(* Logix 5000 project; controller GEA_Test_Chamber vendor 1 type 14 code 196 rev 32.14; software revision 32.04; part 9 of 11 *)
(* tags used below, declared in another part *)
   Act_Time : DINT[7];
   bPulse05Hz : BOOL;
   bPulse0_1Hz : BOOL;
   bPulse10Hz : BOOL;
   bPulse1Hz : BOOL;
   bPulse1min : BOOL;
   Counter : COUNTER[20];
   LDO_LabView_Comm_OK : BOOL;
   LDO_Oil_Step : INT;
   LDO_Step : INT;
   New_Time : BOOL;
   Oil_spray_08_ccmin : BOOL;
   Oil_spray_11_ccmin : BOOL;
   Oil_spray_133_ccmin : BOOL;
   Pulse : BOOL[32];
   Step_10_Done : BOOL;
   Step_20_Done : BOOL;
   Step_25_Done : BOOL;
   Step_30_Done : BOOL;
   Step_40_Done : BOOL;
   Step_5_Done : BOOL;
   T_Diff_10 : DINT;
   T_Diff_20 : DINT;
   T_Diff_25 : DINT;
   T_Diff_30 : DINT;
   T_Diff_40 : DINT;
   T_Diff_5 : DINT;
   T_Diff_Step10 : T_DIFF;
   T_Diff_Step20 : T_DIFF;
   T_Diff_Step25 : T_DIFF;
   T_Diff_Step30 : T_DIFF;
   T_Diff_Step40 : T_DIFF;
   T_Diff_Step5 : T_DIFF;
   Time_Step_10 : DINT[7];
   Time_Step_20 : DINT[7];
   Time_Step_25 : DINT[7];
   Time_Step_30 : DINT[7];
   Time_Step_40 : DINT[7];
   Time_Step_5 : DINT[7];
   tof0_1sPulse : TIMER;
   tof10sPulse : TIMER;
   tof1sPulse : TIMER;
   tof2sPulse : TIMER;
   tof30sPulse : TIMER;
   ton0_1sPulse : TIMER;
   ton10sPulse : TIMER;
   ton1sPulse : TIMER;
   ton2sPulse : TIMER;
   ton30sPulse : TIMER;
   TON_LifeBit_OFF : TIMER;
   TON_LifeBit_ON : TIMER;
   Control_Off : BOOL;
   FVIR_LabView_Control : INT;
   LDO_Error_MSG : INT;
   LDO_LabView_Control : INT;
   LDO_LabView_Control2 : INT;
   LDO_LabView_Status : INT;
   LDO_Reset_CNT_inprogress : BOOL;
   Modbus_LabView_Data : raC_UDT_ModbusServerData;
   Oil_inj_08_Cnt : COUNTER;
   Oil_inj_11_Cnt : COUNTER;
   Oil_inj_133_Cnt : COUNTER;
   Output_LDO : Output_LDO;
(* LDO_Chamber, continued *)

ROUTINE LDO_Main   (* ladder *)
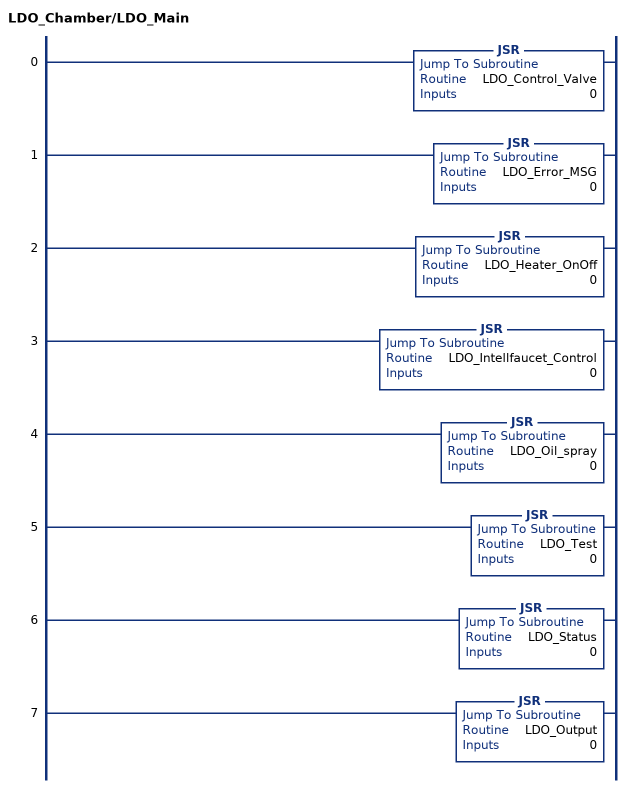
   0: JSR(LDO_Control_Valve,0);
   1: JSR(LDO_Error_MSG,0);
   2: JSR(LDO_Heater_OnOff,0);
   3: JSR(LDO_Intellfaucet_Control,0);
   4: JSR(LDO_Oil_spray,0);
   5: JSR(LDO_Test,0);
   6: JSR(LDO_Status,0);
   7: JSR(LDO_Output,0);
END_ROUTINE

ROUTINE LDO_Oil_spray   (* ladder *)
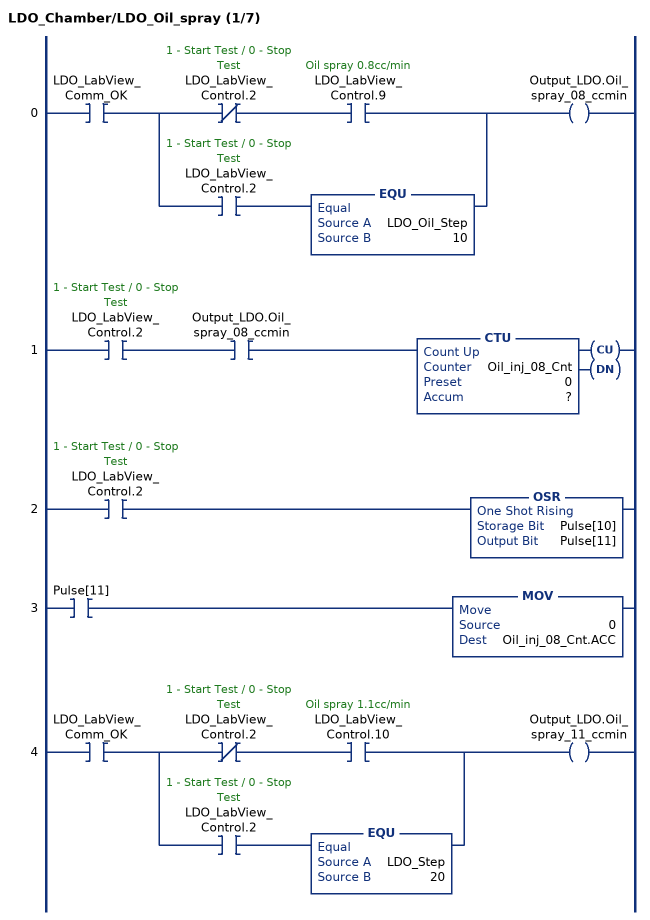
   0: XIC(LDO_LabView_Comm_OK)[XIO(LDO_LabView_Control.2) XIC(LDO_LabView_Control.9) ,XIC(LDO_LabView_Control.2) EQU(LDO_Oil_Step,10) ]OTE(Output_LDO.Oil_spray_08_ccmin);
   1: XIC(LDO_LabView_Control.2)XIC(Output_LDO.Oil_spray_08_ccmin)CTU(Oil_inj_08_Cnt,?,?);
   2: XIC(LDO_LabView_Control.2)OSR(Pulse[10],Pulse[11]);
   3: XIC(Pulse[11])MOV(0,Oil_inj_08_Cnt.ACC);
   4: XIC(LDO_LabView_Comm_OK)[XIO(LDO_LabView_Control.2) XIC(LDO_LabView_Control.10) ,XIC(LDO_LabView_Control.2) EQU(LDO_Step,20) ]OTE(Output_LDO.Oil_spray_11_ccmin);
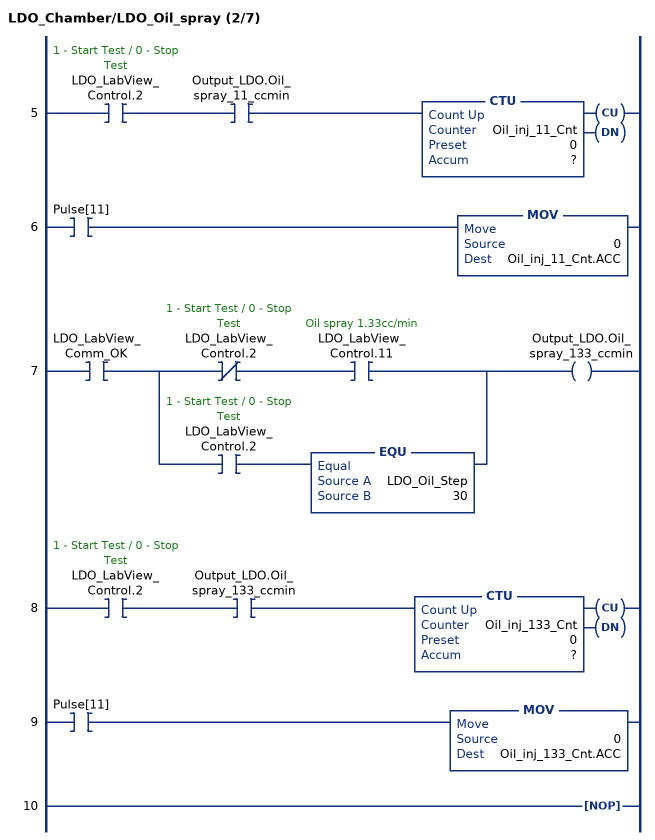
   5: XIC(LDO_LabView_Control.2)XIC(Output_LDO.Oil_spray_11_ccmin)CTU(Oil_inj_11_Cnt,?,?);
   6: XIC(Pulse[11])MOV(0,Oil_inj_11_Cnt.ACC);
   7: XIC(LDO_LabView_Comm_OK)[XIO(LDO_LabView_Control.2) XIC(LDO_LabView_Control.11) ,XIC(LDO_LabView_Control.2) EQU(LDO_Oil_Step,30) ]OTE(Output_LDO.Oil_spray_133_ccmin);
   8: XIC(LDO_LabView_Control.2)XIC(Output_LDO.Oil_spray_133_ccmin)CTU(Oil_inj_133_Cnt,?,?);
   9: XIC(Pulse[11])MOV(0,Oil_inj_133_Cnt.ACC);
   10: NOP();
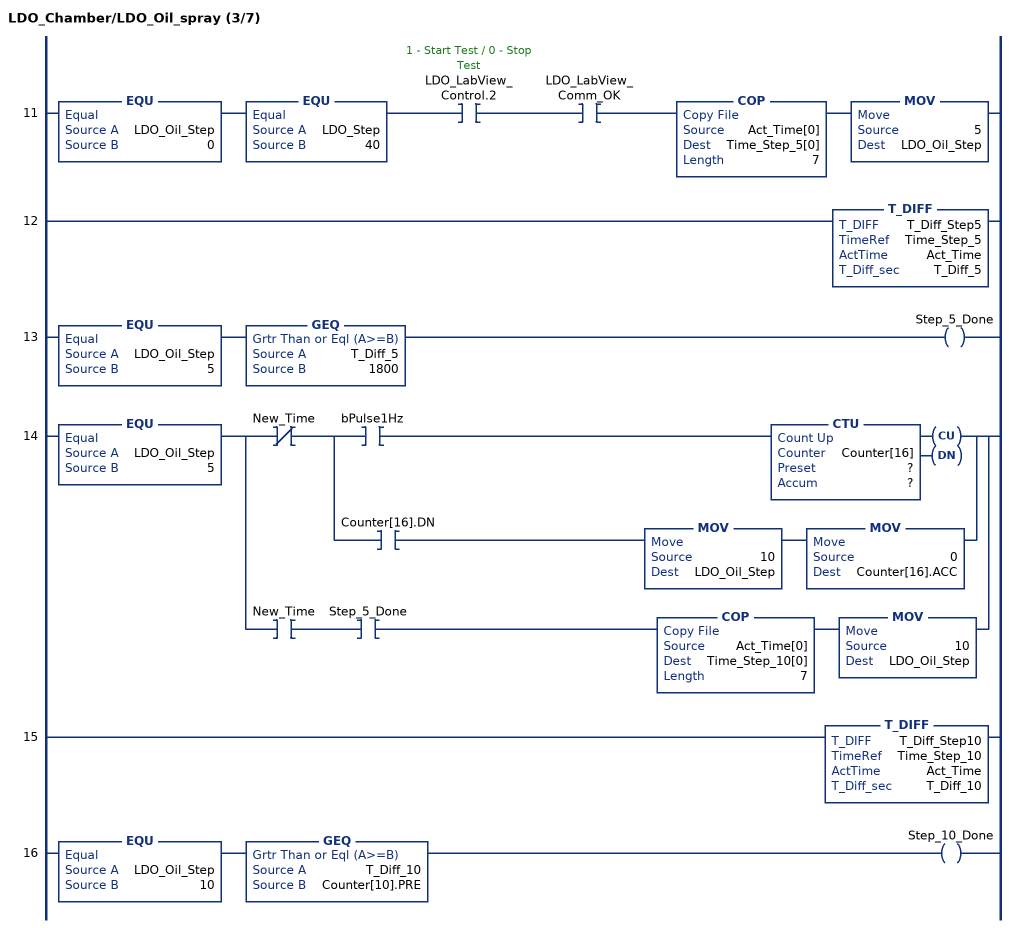
   11: EQU(LDO_Oil_Step,0)EQU(LDO_Step,40)XIC(LDO_LabView_Control.2)XIC(LDO_LabView_Comm_OK)COP(Act_Time[0],Time_Step_5[0],7)MOV(5,LDO_Oil_Step);
   12: T_DIFF(T_Diff_Step5,Time_Step_5,Act_Time,T_Diff_5);
   13: EQU(LDO_Oil_Step,5)GEQ(T_Diff_5,1800)OTE(Step_5_Done);
   14: EQU(LDO_Oil_Step,5)[XIO(New_Time) [XIC(bPulse1Hz) CTU(Counter[16],?,?) ,XIC(Counter[16].DN) MOV(10,LDO_Oil_Step) MOV(0,Counter[16].ACC) ] ,XIC(New_Time) XIC(Step_5_Done) COP(Act_Time[0],Time_Step_10[0],7) MOV(10,LDO_Oil_Step) ];
   15: T_DIFF(T_Diff_Step10,Time_Step_10,Act_Time,T_Diff_10);
   16: EQU(LDO_Oil_Step,10)GEQ(T_Diff_10,Counter[10].PRE)OTE(Step_10_Done);
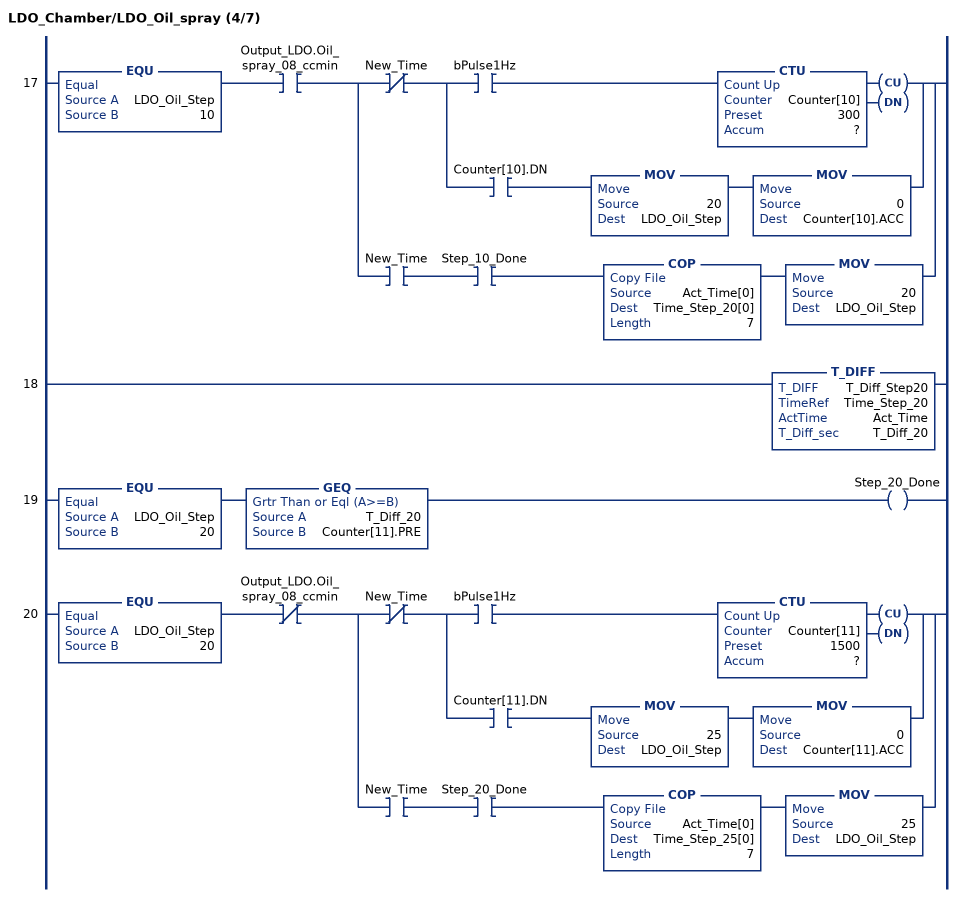
   17: EQU(LDO_Oil_Step,10)XIC(Output_LDO.Oil_spray_08_ccmin)[XIO(New_Time) [XIC(bPulse1Hz) CTU(Counter[10],?,?) ,XIC(Counter[10].DN) MOV(20,LDO_Oil_Step) MOV(0,Counter[10].ACC) ] ,XIC(New_Time) XIC(Step_10_Done) COP(Act_Time[0],Time_Step_20[0],7) MOV(20,LDO_Oil_Step) ];
   18: T_DIFF(T_Diff_Step20,Time_Step_20,Act_Time,T_Diff_20);
   19: EQU(LDO_Oil_Step,20)GEQ(T_Diff_20,Counter[11].PRE)OTE(Step_20_Done);
   20: EQU(LDO_Oil_Step,20)XIO(Output_LDO.Oil_spray_08_ccmin)[XIO(New_Time) [XIC(bPulse1Hz) CTU(Counter[11],?,?) ,XIC(Counter[11].DN) MOV(25,LDO_Oil_Step) MOV(0,Counter[11].ACC) ] ,XIC(New_Time) XIC(Step_20_Done) COP(Act_Time[0],Time_Step_25[0],7) MOV(25,LDO_Oil_Step) ];
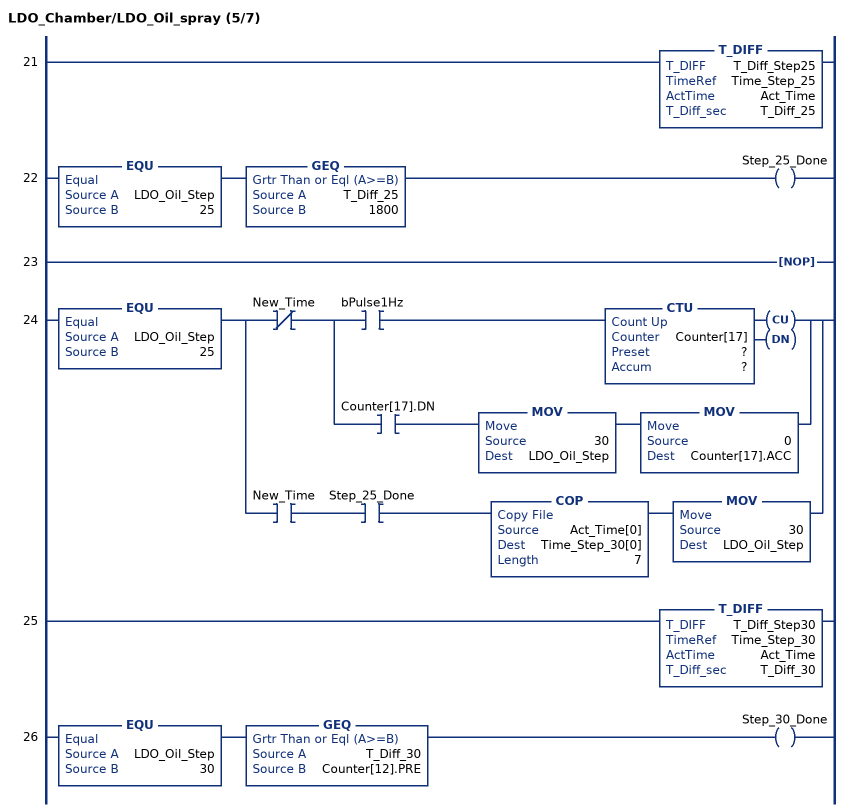
   21: T_DIFF(T_Diff_Step25,Time_Step_25,Act_Time,T_Diff_25);
   22: EQU(LDO_Oil_Step,25)GEQ(T_Diff_25,1800)OTE(Step_25_Done);
   23: NOP();
   24: EQU(LDO_Oil_Step,25)[XIO(New_Time) [XIC(bPulse1Hz) CTU(Counter[17],?,?) ,XIC(Counter[17].DN) MOV(30,LDO_Oil_Step) MOV(0,Counter[17].ACC) ] ,XIC(New_Time) XIC(Step_25_Done) COP(Act_Time[0],Time_Step_30[0],7) MOV(30,LDO_Oil_Step) ];
   25: T_DIFF(T_Diff_Step30,Time_Step_30,Act_Time,T_Diff_30);
   26: EQU(LDO_Oil_Step,30)GEQ(T_Diff_30,Counter[12].PRE)OTE(Step_30_Done);
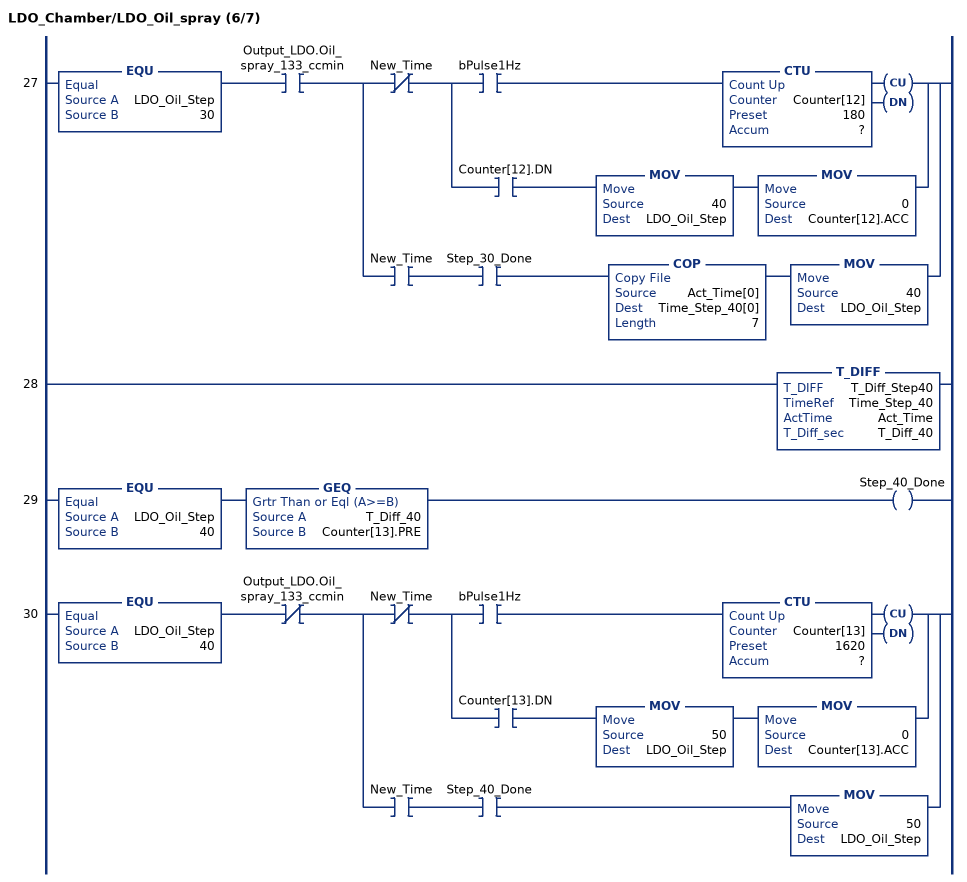
   27: EQU(LDO_Oil_Step,30)XIC(Output_LDO.Oil_spray_133_ccmin)[XIO(New_Time) [XIC(bPulse1Hz) CTU(Counter[12],?,?) ,XIC(Counter[12].DN) MOV(40,LDO_Oil_Step) MOV(0,Counter[12].ACC) ] ,XIC(New_Time) XIC(Step_30_Done) COP(Act_Time[0],Time_Step_40[0],7) MOV(40,LDO_Oil_Step) ];
   28: T_DIFF(T_Diff_Step40,Time_Step_40,Act_Time,T_Diff_40);
   29: EQU(LDO_Oil_Step,40)GEQ(T_Diff_40,Counter[13].PRE)OTE(Step_40_Done);
   30: EQU(LDO_Oil_Step,40)XIO(Output_LDO.Oil_spray_133_ccmin)[XIO(New_Time) [XIC(bPulse1Hz) CTU(Counter[13],?,?) ,XIC(Counter[13].DN) MOV(50,LDO_Oil_Step) MOV(0,Counter[13].ACC) ] ,XIC(New_Time) XIC(Step_40_Done) MOV(50,LDO_Oil_Step) ];
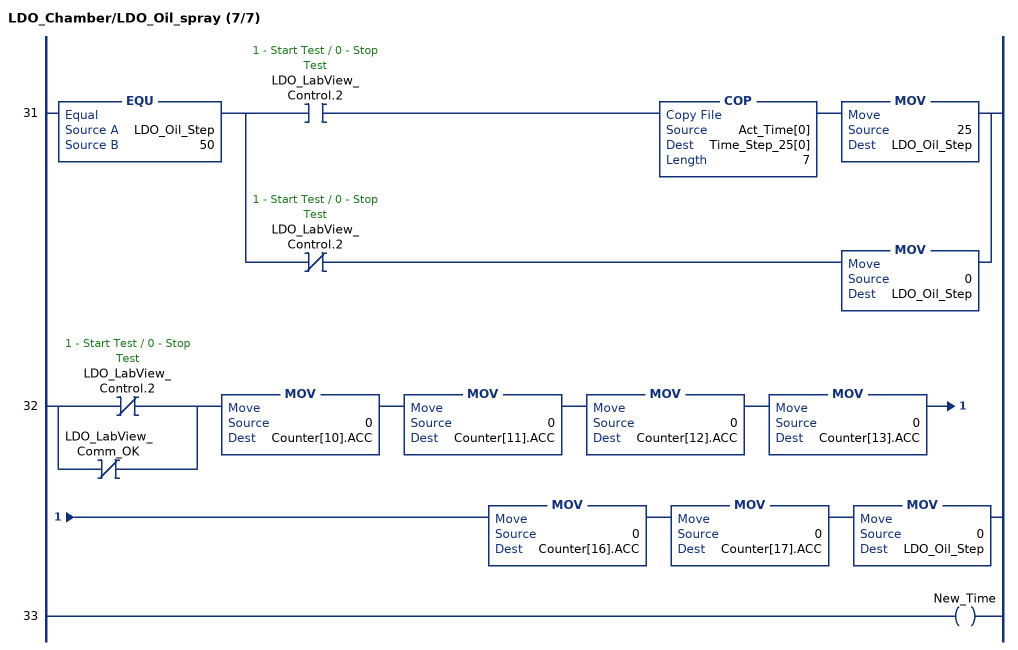
   31: EQU(LDO_Oil_Step,50)[XIC(LDO_LabView_Control.2) COP(Act_Time[0],Time_Step_25[0],7) MOV(25,LDO_Oil_Step) ,XIO(LDO_LabView_Control.2) MOV(0,LDO_Oil_Step) ];
   32: [XIO(LDO_LabView_Control.2) ,XIO(LDO_LabView_Comm_OK) ]MOV(0,Counter[10].ACC)MOV(0,Counter[11].ACC)MOV(0,Counter[12].ACC)MOV(0,Counter[13].ACC)MOV(0,Counter[16].ACC)MOV(0,Counter[17].ACC)MOV(0,LDO_Oil_Step);
   33: OTE(New_Time);
END_ROUTINE

ROUTINE LDO_Output   (* ladder *)
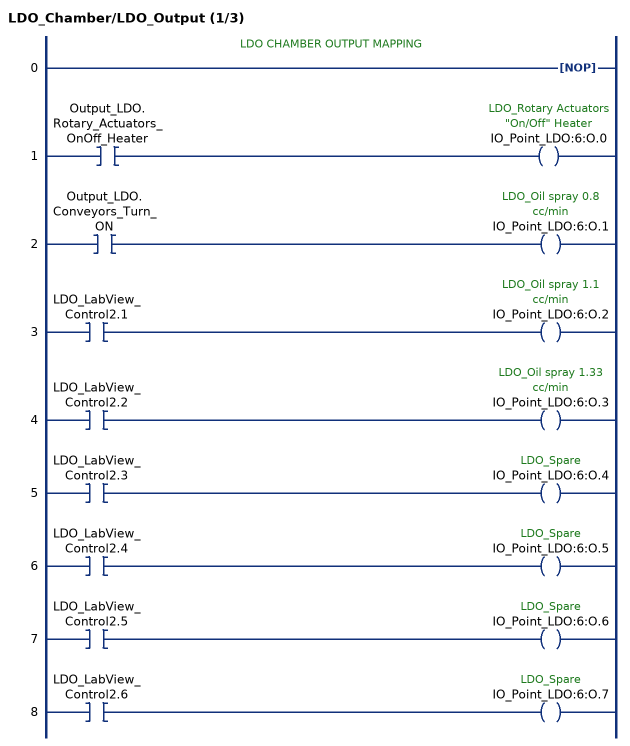
   // LDO CHAMBER OUTPUT MAPPING
   0: NOP();
   1: XIC(Output_LDO.Rotary_Actuators_OnOff_Heater)OTE(IO_Point_LDO:6:O.0);
   2: XIC(Output_LDO.Conveyors_Turn_ON)OTE(IO_Point_LDO:6:O.1);
   3: XIC(LDO_LabView_Control2.1)OTE(IO_Point_LDO:6:O.2);
   4: XIC(LDO_LabView_Control2.2)OTE(IO_Point_LDO:6:O.3);
   5: XIC(LDO_LabView_Control2.3)OTE(IO_Point_LDO:6:O.4);
   6: XIC(LDO_LabView_Control2.4)OTE(IO_Point_LDO:6:O.5);
   7: XIC(LDO_LabView_Control2.5)OTE(IO_Point_LDO:6:O.6);
   8: XIC(LDO_LabView_Control2.6)OTE(IO_Point_LDO:6:O.7);
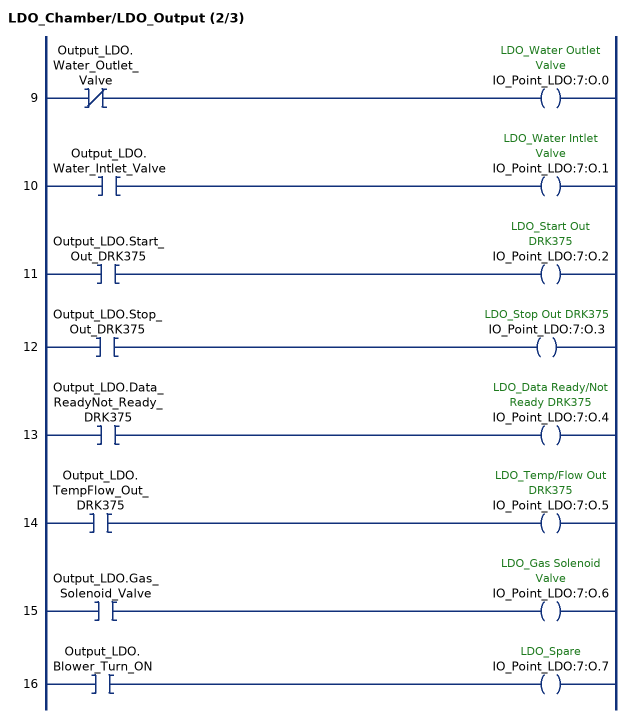
   9: XIO(Output_LDO.Water_Outlet_Valve)OTE(IO_Point_LDO:7:O.0);
   10: XIC(Output_LDO.Water_Intlet_Valve)OTE(IO_Point_LDO:7:O.1);
   11: XIC(Output_LDO.Start_Out_DRK375)OTE(IO_Point_LDO:7:O.2);
   12: XIC(Output_LDO.Stop_Out_DRK375)OTE(IO_Point_LDO:7:O.3);
   13: XIC(Output_LDO.Data_ReadyNot_Ready_DRK375)OTE(IO_Point_LDO:7:O.4);
   14: XIC(Output_LDO.TempFlow_Out_DRK375)OTE(IO_Point_LDO:7:O.5);
   15: XIC(Output_LDO.Gas_Solenoid_Valve)OTE(IO_Point_LDO:7:O.6);
   16: XIC(Output_LDO.Blower_Turn_ON)OTE(IO_Point_LDO:7:O.7);
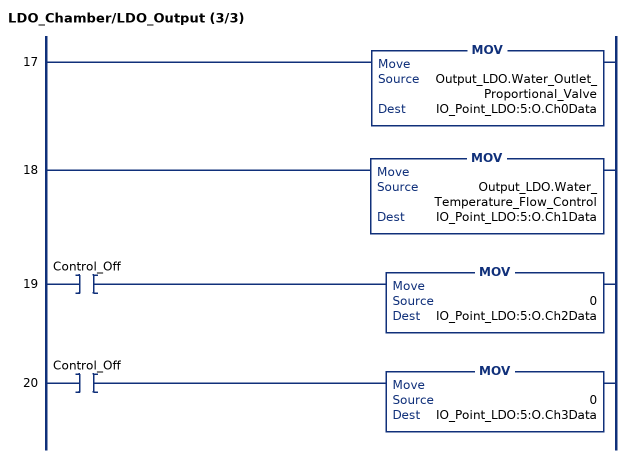
   17: MOV(Output_LDO.Water_Outlet_Proportional_Valve,IO_Point_LDO:5:O.Ch0Data);
   18: MOV(Output_LDO.Water_Temperature_Flow_Control,IO_Point_LDO:5:O.Ch1Data);
   19: XIC(Control_Off)MOV(0,IO_Point_LDO:5:O.Ch2Data);
   20: XIC(Control_Off)MOV(0,IO_Point_LDO:5:O.Ch3Data);
END_ROUTINE

ROUTINE LDO_Status   (* ladder *)
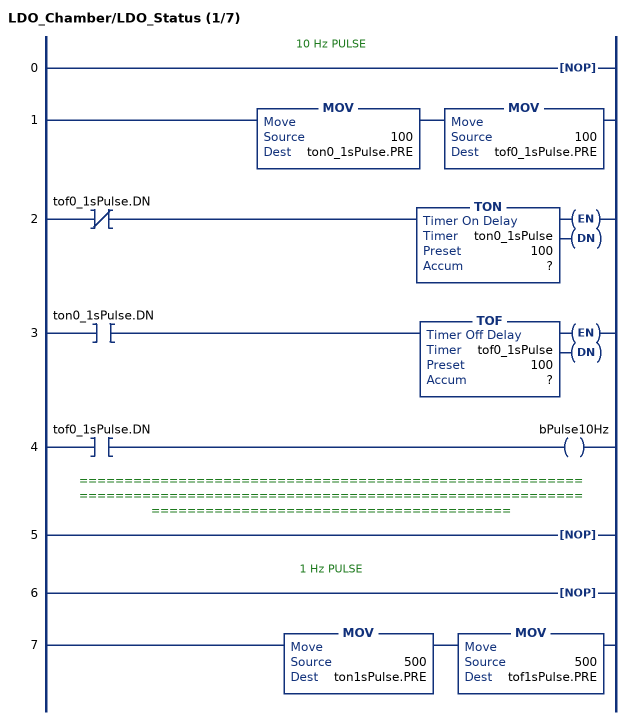
   // 10 Hz PULSE
   0: NOP();
   1: MOV(100,ton0_1sPulse.PRE)MOV(100,tof0_1sPulse.PRE);
   2: XIO(tof0_1sPulse.DN)TON(ton0_1sPulse,?,?);
   3: XIC(ton0_1sPulse.DN)TOF(tof0_1sPulse,?,?);
   4: XIC(tof0_1sPulse.DN)OTE(bPulse10Hz);
   // ========================================================================================================================================================
   5: NOP();
   // 1 Hz PULSE
   6: NOP();
   7: MOV(500,ton1sPulse.PRE)MOV(500,tof1sPulse.PRE);
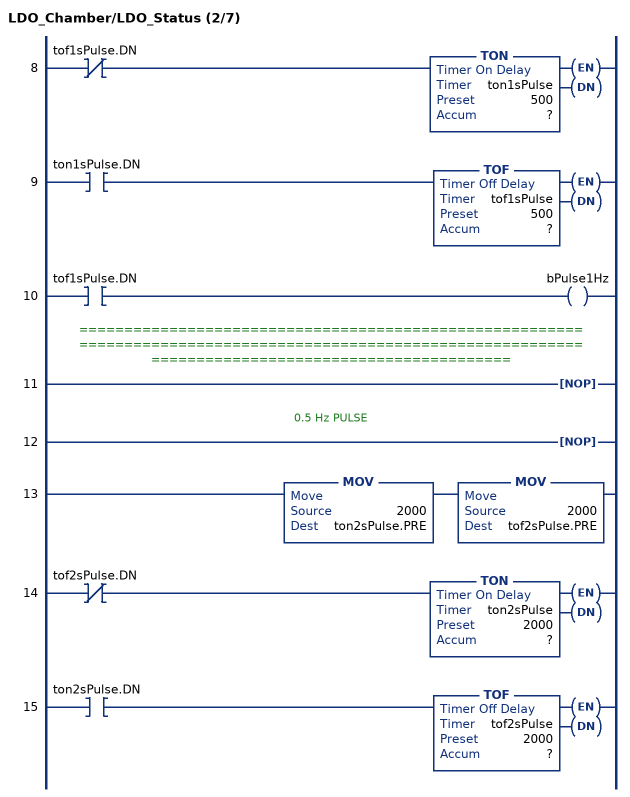
   8: XIO(tof1sPulse.DN)TON(ton1sPulse,?,?);
   9: XIC(ton1sPulse.DN)TOF(tof1sPulse,?,?);
   10: XIC(tof1sPulse.DN)OTE(bPulse1Hz);
   // ========================================================================================================================================================
   11: NOP();
   // 0.5 Hz PULSE
   12: NOP();
   13: MOV(2000,ton2sPulse.PRE)MOV(2000,tof2sPulse.PRE);
   14: XIO(tof2sPulse.DN)TON(ton2sPulse,?,?);
   15: XIC(ton2sPulse.DN)TOF(tof2sPulse,?,?);
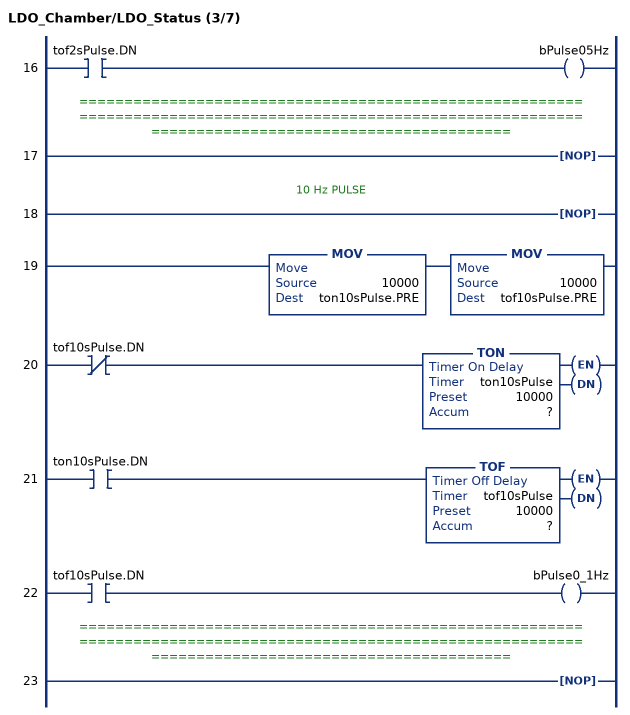
   16: XIC(tof2sPulse.DN)OTE(bPulse05Hz);
   // ========================================================================================================================================================
   17: NOP();
   // 10 Hz PULSE
   18: NOP();
   19: MOV(10000,ton10sPulse.PRE)MOV(10000,tof10sPulse.PRE);
   20: XIO(tof10sPulse.DN)TON(ton10sPulse,?,?);
   21: XIC(ton10sPulse.DN)TOF(tof10sPulse,?,?);
   22: XIC(tof10sPulse.DN)OTE(bPulse0_1Hz);
   // ========================================================================================================================================================
   23: NOP();
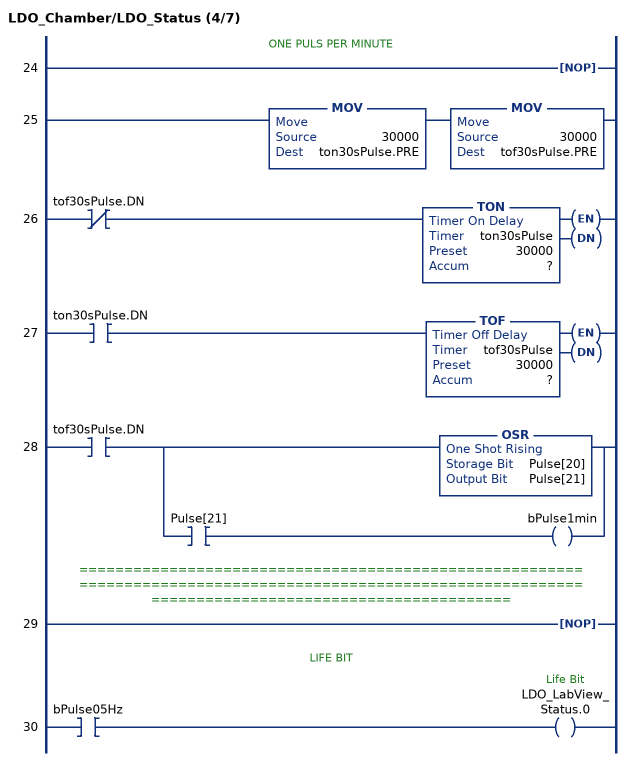
   // ONE PULS PER MINUTE
   24: NOP();
   25: MOV(30000,ton30sPulse.PRE)MOV(30000,tof30sPulse.PRE);
   26: XIO(tof30sPulse.DN)TON(ton30sPulse,?,?);
   27: XIC(ton30sPulse.DN)TOF(tof30sPulse,?,?);
   28: XIC(tof30sPulse.DN)[OSR(Pulse[20],Pulse[21]) ,XIC(Pulse[21]) OTE(bPulse1min) ];
   // ========================================================================================================================================================
   29: NOP();
   // LIFE BIT
   30: XIC(bPulse05Hz)OTE(LDO_LabView_Status.0);
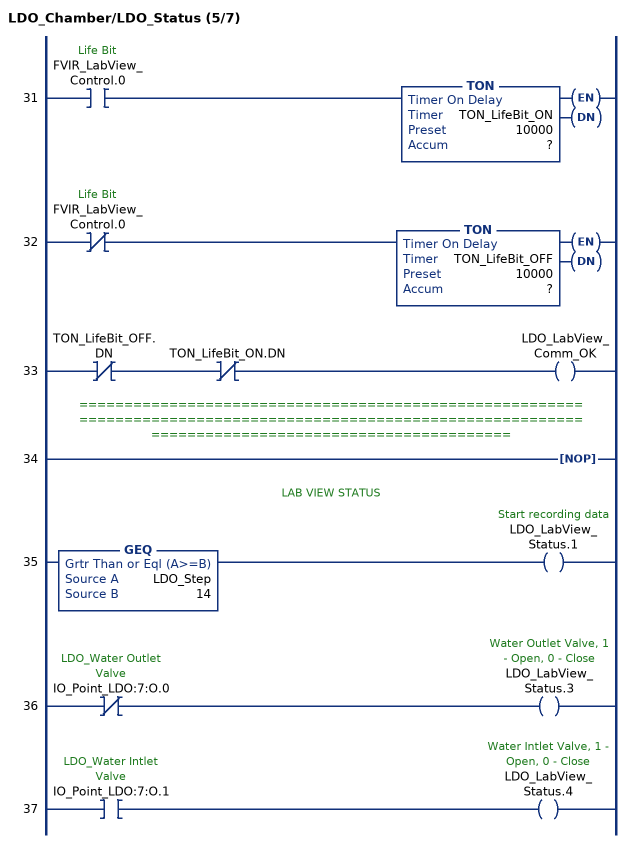
   31: XIC(FVIR_LabView_Control.0)TON(TON_LifeBit_ON,?,?);
   32: XIO(FVIR_LabView_Control.0)TON(TON_LifeBit_OFF,?,?);
   33: XIO(TON_LifeBit_OFF.DN)XIO(TON_LifeBit_ON.DN)OTE(LDO_LabView_Comm_OK);
   // ========================================================================================================================================================
   34: NOP();
   // LAB VIEW STATUS
   35: GEQ(LDO_Step,14)OTE(LDO_LabView_Status.1);
   36: XIO(IO_Point_LDO:7:O.0)OTE(LDO_LabView_Status.3);
   37: XIC(IO_Point_LDO:7:O.1)OTE(LDO_LabView_Status.4);
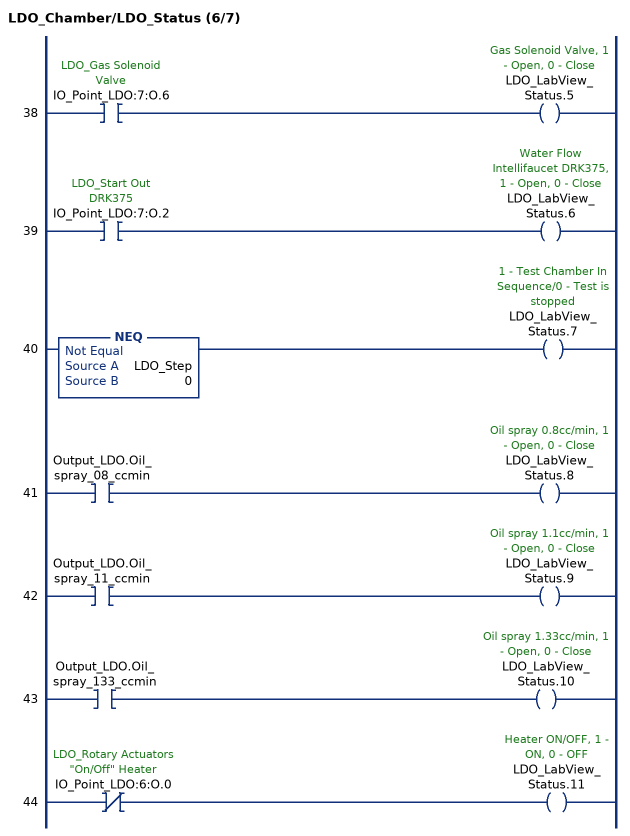
   38: XIC(IO_Point_LDO:7:O.6)OTE(LDO_LabView_Status.5);
   39: XIC(IO_Point_LDO:7:O.2)OTE(LDO_LabView_Status.6);
   40: NEQ(LDO_Step,0)OTE(LDO_LabView_Status.7);
   41: XIC(Output_LDO.Oil_spray_08_ccmin)OTE(LDO_LabView_Status.8);
   42: XIC(Output_LDO.Oil_spray_11_ccmin)OTE(LDO_LabView_Status.9);
   43: XIC(Output_LDO.Oil_spray_133_ccmin)OTE(LDO_LabView_Status.10);
   44: XIO(IO_Point_LDO:6:O.0)OTE(LDO_LabView_Status.11);
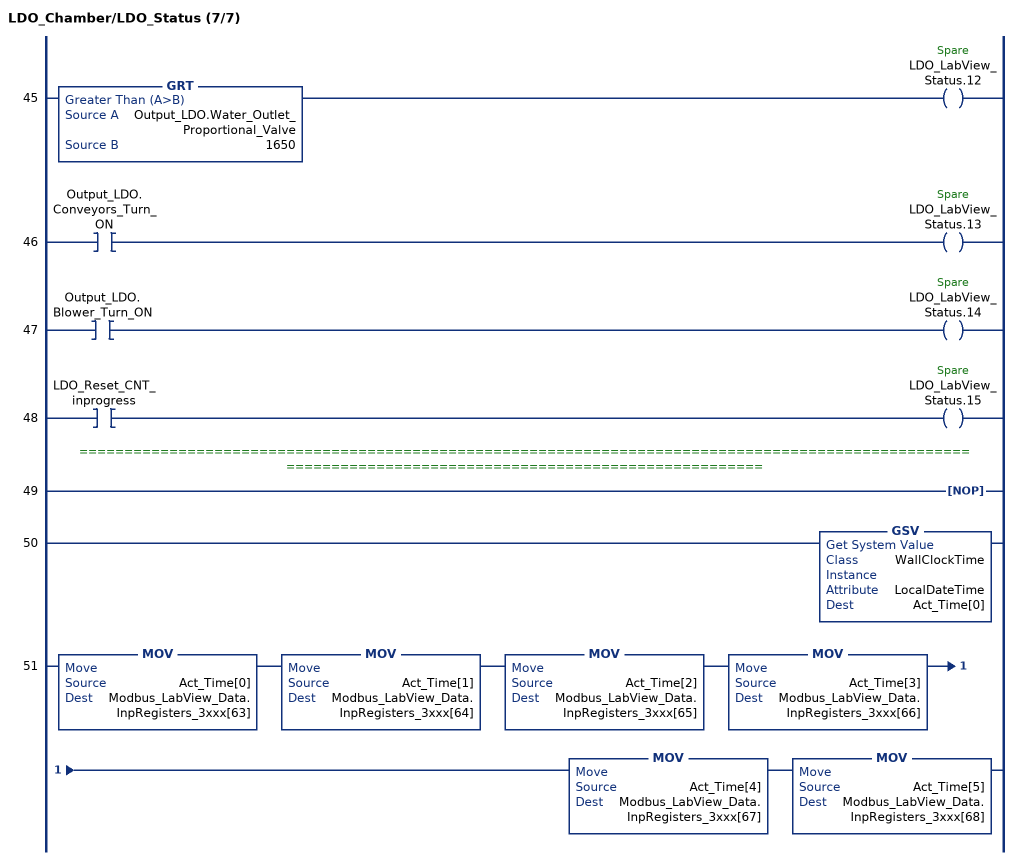
   45: GRT(Output_LDO.Water_Outlet_Proportional_Valve,1650)OTE(LDO_LabView_Status.12);
   46: XIC(Output_LDO.Conveyors_Turn_ON)OTE(LDO_LabView_Status.13);
   47: XIC(Output_LDO.Blower_Turn_ON)OTE(LDO_LabView_Status.14);
   48: XIC(LDO_Reset_CNT_inprogress)OTE(LDO_LabView_Status.15);
   // ========================================================================================================================================================
   49: NOP();
   50: GSV(WallClockTime,,LocalDateTime,Act_Time[0]);
   51: MOV(Act_Time[0],Modbus_LabView_Data.InpRegisters_3xxx[63])MOV(Act_Time[1],Modbus_LabView_Data.InpRegisters_3xxx[64])MOV(Act_Time[2],Modbus_LabView_Data.InpRegisters_3xxx[65])MOV(Act_Time[3],Modbus_LabView_Data.InpRegisters_3xxx[66])MOV(Act_Time[4],Modbus_LabView_Data.InpRegisters_3xxx[67])MOV(Act_Time[5],Modbus_LabView_Data.InpRegisters_3xxx[68]);
END_ROUTINE
